// TwinCAT 3 PLC project Ben_Harrison_Prototype
// ProgramVersion: 3.1.4024.0
// libraries:
//   Tc2_Standard, * (Beckhoff Automation GmbH)
//   Tc2_System, * (Beckhoff Automation GmbH)
//   Tc3_Module, * (Beckhoff Automation GmbH)
// project tree:
//   / Class Diagram_3.TcCD (not stored), Class Diagram_8.TcCD (not stored), PlcTask.TcTTO (not stored)
//   Classes/ Circle.TcPOU (not stored), Disposable.TcPOU (not stored), Rectangle.TcPOU (not stored)
//   Interfaces/ I_Disposable.TcIO (not stored), I_DrawableShape.TcIO (not stored)
//   POUs/ MAIN.TcPOU
// real-time tasks:
//   TASK PlcTask: cycle T#10ms, priority 20, ADS port 350

// ---- POUs/MAIN.TcPOU
PROGRAM MAIN
VAR
    originalRectangle: Rectangle;
    clonedRectangle: I_DrawableShape;
	
    originalCircle: Circle;
    clonedCircle: I_DrawableShape;
	
	bRequest : BOOL;
	counter: INT;

END_VAR

// https://refactoring.guru/design-patterns/prototype

// Recuerda que el patrón Prototipo permite crear nuevos objetos clonando un objeto existente, evitando así la necesidad de crear nuevas instancias desde cero.

// porque salen varios mensajes:
// https://github.com/tcunit/TcUnit/issues/92
// solución temporal : Unload project...
IF bRequest THEN
	
	// rectangle example 
	originalRectangle.Width := 10;
	originalRectangle.Height := 5;
	originalRectangle.Draw();
	clonedRectangle := originalRectangle.clone();
	clonedRectangle.Draw();
	clonedRectangle.Dispose(); 
	
	// circle example 
	originalCircle.Radius := 7;
	originalCircle.Draw();
	clonedCircle := originalCircle.clone();
	clonedCircle.Draw();
	clonedCircle.Dispose(); 
	
	// report request info
	bRequest := FALSE;
	counter := counter + 1;
	ADSLOGSTR(msgCtrlMask :=ADSLOG_MSGTYPE_HINT, msgFmtStr :='test: %s', strArg := TO_STRING(counter));

END_IF

END_PROGRAM
